FUNCTION_BLOCK FB_Module02 EXTENDS FB_Module
VAR_INPUT
END_VAR
VAR_OUTPUT
END_VAR
VAR
	fbPnozMulti:				FB_PnozMulti;
	fbComponent0:				FB_ComponentEx;
	fbComponent1:				FB_ComponentEx;
	fbContactor:				FB_Contactor;
	fbCylinder:					FB_Cylinder;
END_VAR

// https://peterzerlauth.com/
SUPER^();

fbComponent0();
fbComponent1();
fbContactor();
fbCylinder();
fbPnozMulti();

fbContactor.bInput:= fbContactor.bOutput;

METHOD PROTECTED M_Execute : BOOL
VAR_INPUT
END_VAR
VAR
	bReturn:					BOOL:= TRUE;
END_VAR
CASE fbSequence.P_Number OF
	E_Sequence.Start:
		bReturn:= TRUE;
		fbSequence.M_Await('Start 0', 0,  T#0S , T#1S, TRUE, bReturn, 10);
	
	10:
		bReturn:= TRUE;
		fbSequence.M_Await('Step 10', 0,  T#0S, T#0S, TRUE, bReturn, 20);
		
	20:
		bReturn:= TRUE;
		fbSequence.M_Await('Step 20', 0,  T#1S, T#0S, FALSE, bReturn, E_Sequence.Done);
		IF fbSequence.P_Timeout THEN
			fbEvent.M_Error('Overrride timeout error', 0);
		END_IF
		
	E_Sequence.Done:
		fbSequence.M_Reset();

END_CASE
END_METHOD

METHOD PROTECTED M_Idle : BOOL (* Return*)
SUPER^.M_Idle();

fbLevel2.M_Attach(fbPnozMulti);
fbLevel2.M_Attach(fbComponent0);
fbLevel2.M_Attach(fbComponent1);
fbLevel2.M_Attach(fbPnozMulti);
fbLevel2.M_Attach(fbContactor);
fbLevel1.M_Attach(fbCylinder);
END_METHOD

END_FUNCTION_BLOCK

(* stored: Version 1.1.0.1
   POU FB_Module02: Id {c6d30f55-be05-0005-0105-ea54e786664b}, SpecialFunc None
   Method M_Execute: Id {06feba3b-22b0-0914-2021-212ac5c61859}
   Method M_Idle: Id {68b2e8eb-c718-0ade-0688-6a32403d9271} *)
